PROGRAM PRG_1_PlcTask
VAR
END_VAR

PRG_2_PMPS_PRE();

PRG_IM1K0_XTES();
PRG_IM1K3_PPM();
PRG_IM2K0_XTES();
PRG_PF1K0_WFS();
PRG_RTDSK0();
PRG_SL1K0_POWER();
PRG_SL2K0_POWER();

PRG_AT1K4_SOLID();
PRG_IM1K4_XTES();
PRG_ST1K4_TEST();
PRG_OTHER();

PRG_3_PMPS_POST();
PRG_4_LOG();

END_PROGRAM

(* stored: Version 1.1.0.1, ProductVersion 3.1.4022.18
   POU PRG_1_PlcTask: Id {b12fe210-df04-4a98-819b-8df554fce2a7}, SpecialFunc None *)
